{attribute 'qualified_only'}
VAR_GLOBAL
	position: UINT := 0;
	velocity: UINT := 0;
	acceleration: UINT := 0;
	execute: BOOL := FALSE;
END_VAR

(* stored: Version 1.1.0.1, ProductVersion 3.1.4024.12
   GVL GVL_VARS2: Id {ee2c1af7-fa8d-4cfa-a856-8093e932e508} *)
